(* CoDeSys 2.3.9.47 project: incomplete parking.pro *)
(* Libraries: Nexgenie.lib*28.8.18 12:27:24, Standard.lib*28.8.18 12:27:25, Nexgenie_Util.lib*28.8.18 12:27:24, Nexgenie_H.lib*28.8.18 12:27:24, VAW.lib*28.8.18 12:27:25, Modbus.lib*28.8.18 12:27:24 *)

(* PLC configuration (modules and I/O channels)
Nexgenie1000 [Root] node -1, in %IB0 out %QB0
  Nexgenie [Nexgenie] node 0, in %IB0 out %QB0
*)

(* POU PLC_PRG, LD *)
PROGRAM PLC_PRG
VAR
	entry: BOOL;
	stop: BOOL;
	c_sec: CTU;
	X1: BOOL;
	x2: BOOL;
	d_sec: INT;
	A_sec: INT;
END_VAR
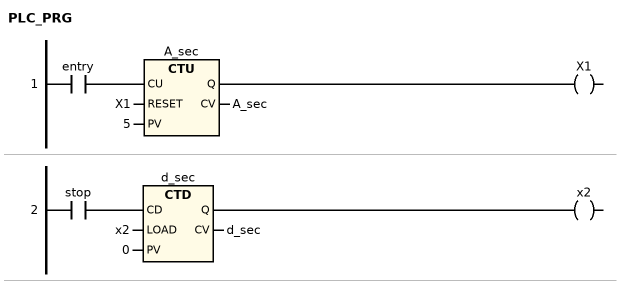
_LD_ (* Ladder Diagram *)
NETWORK 1
	[entry] - A_sec:CTU(CU: *, RESET: X1, PV: 5, CV => A_sec) --- (X1)
NETWORK 2
	[stop] - d_sec:CTD(CD: *, LOAD: x2, PV: 0, CV => d_sec) --- (x2)
_END_LD_
(* the same logic as Structured Text *)
(* Network 1 *)
A_sec(CU := entry, RESET := X1, PV := 5);
A_sec := A_sec.CV;
X1 := A_sec.Q;
(* Network 2 *)
d_sec(CD := stop, LOAD := x2, PV := 0);
d_sec := d_sec.CV;
x2 := d_sec.Q;
END_PROGRAM

(* Visualisation LOL
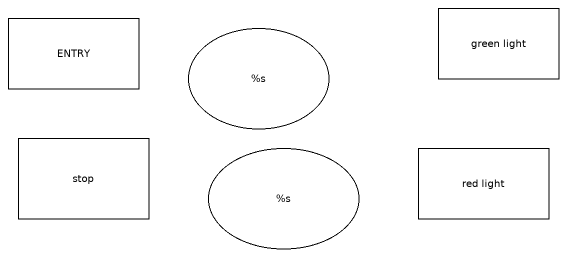
rectangle at (30,60)-(161,131): text "ENTRY"; alarm colour if PLC_PRG.entry; toggles PLC_PRG.entry
rectangle at (460,50)-(581,121): text "green light"; alarm colour if PLC_PRG.X1
rectangle at (40,180)-(171,261): text "stop"; alarm colour if PLC_PRG.stop; toggles PLC_PRG.stop
rectangle at (440,190)-(571,261): text "red light"; alarm colour if PLC_PRG.x2
ellipse at (210,70)-(351,171): text "%s"; shows PLC_PRG.A_sec
ellipse at (230,190)-(381,291): text "%s"; shows PLC_PRG.
*)
